{attribute addProperty BoxType "EK1960-2600-0019"}
{attribute addProperty Id "FSoE_InputsFSoE_Inputs_0C161FF712015FSoE_OutputsFSoE_Outputs_E86FAAD612015"}
{attribute addProperty CRC "3659517265"}
{attribute addProperty SizeInBites "240"}
{attribute addProperty SizeInBytes "30"}
TYPE Module_1_FSoE_DA1FCD51 :
STRUCT
	{attribute addProperty Name "FSoE_Inputs"}
	FSoE_Inputs  : FSoE_Inputs_0C161FF7;
	{attribute addProperty Name "FSoE_Outputs"}
	FSoE_Outputs  : FSoE_Outputs_E86FAAD6;
END_STRUCT
END_TYPE

(* stored: Version 1.2.0.0, ProductVersion 3.1.4024.9
   DUT Module_1_FSoE_DA1FCD51: Id {6e94a216-c8f2-4900-af13-d2eb86d5a856} *)
